TYPE SliderAttenuationFilterConfigs :
STRUCT
	ELL6SliderFilterConfig : ELL6AttenuationFilterConfig;
END_STRUCT
END_TYPE

(* stored: Version 1.1.0.1, ProductVersion 3.1.4024.10
   DUT SliderAttenuationFilterConfigs: Id {99ac46d8-de52-4c67-9b89-8aa24c4c8b48} *)
